Omron CX-Programmer project NewProject (CX-Programmer 9.70)

# PLC NewPLC1: CP1E E20

## Global symbols (name address type ; comment)
0.00 BOOL  ; pb on
0.03 BOOL  ; pb2 on
0.04 BOOL  ; pb2 off
10.00 BOOL  ; motor
10.01 BOOL  ; motor2

## Program NewProgram1 (cyclic task 0)
Local symbols
nc 0.01 BOOL  ; pb off

### Section Section1

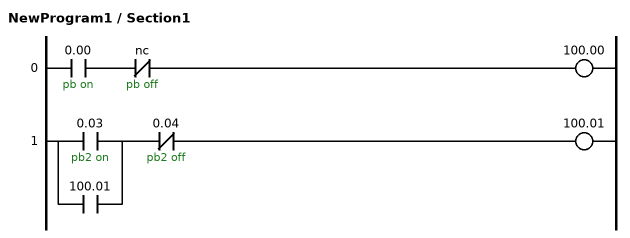
; rung 0
LD 0.00  ; pb on
ANDNOT nc  ; pb off
OUT 100.00
; rung 1
LD 0.03  ; pb2 on
OR 100.01
ANDNOT 0.04  ; pb2 off
OUT 100.01
; rung 2
END(001)

### Section END
; rung 0
END(001)